{attribute addProperty BoxType "CU1128--0000"}
{attribute addProperty Id "A_0005_CU1128_0000_0001A_0005_CU1128_0000_0001_15602991918114.75A_0004_CU1128_0000_0000_2_CU1128_BCU1128_179A0949162A_0004_CU1128_0000_0000_3_CU1128_CCU1128_179A0949162"}
{attribute addProperty CRC "3765028164"}
{attribute addProperty SizeInBites "950"}
{attribute addProperty SizeInBytes "118.75"}
TYPE A_0004_CU1128_0000_0000_E069C544 EXTENDS CU1128_179A0949 :
STRUCT
	{attribute addProperty Name "A_0005_CU1128_0000_0001"}
	A_0005_CU1128_0000_0001 : A_0005_CU1128_0000_0001_15602991;
	{attribute addProperty Name "A_0004_CU1128_0000_0000_2_CU1128_B"}
	A_0004_CU1128_0000_0000_2_CU1128_B : CU1128_179A0949;
	{attribute addProperty Name "A_0004_CU1128_0000_0000_3_CU1128_C"}
	A_0004_CU1128_0000_0000_3_CU1128_C : CU1128_179A0949;
END_STRUCT
END_TYPE

(* stored: Version 1.2.0.0, ProductVersion 3.1.4024.9
   DUT A_0004_CU1128_0000_0000_E069C544: Id {470747d9-2cb9-4032-8dab-a319c2ea9930} *)
